TYPE ST_PLCGroupSetAxis :
STRUCT
	
	st_EachSetAxis : ARRAY [0..19] OF ST_PLCSetAxis;

END_STRUCT
END_TYPE

(* stored: Version 1.1.0.1, ProductVersion 3.1.4022.12
   DUT ST_PLCGroupSetAxis: Id {6dcec074-6a04-4650-930e-118e43e0037e} *)
